(* PLC project variable_speed_drive, Dassault Systèmes ControlBuild 2024x *)
(* stored: creationDateTime 2023-10-03T11:13:08-01:00 *)

(* This module simulates the behaviour of a motor, its variable speed drive and its electrical control logic. The speed setpoint can go from -100% to +100%. *)
FUNCTION_BLOCK equipment_library.variable_speed_drive
  VAR_INPUT
    voltage380 : BOOL := true;
    cmdSupply : BOOL := true;
    sensorSupply : BOOL := true;
  END_VAR
  VAR_INPUT
    forward : BOOL := false;
    speedSetpoint : REAL := 0.0;
  END_VAR
  VAR_OUTPUT
    forwardFB : BOOL := false;
    thermal : BOOL := false;
  END_VAR
  VAR_OUTPUT
    speedVal : REAL := 0.0;
    speedPercent : REAL := 0.0;
  END_VAR
  VAR
    increment : REAL := 0.0;
    memoFwd : BOOL := false;
    forwardState : BOOL := false;
    wantedSpeed : REAL := 0.0;
  END_VAR
  VAR CONSTANT
    nominalSpeed : REAL := 5000.0;
    nominalTime : REAL := 0.5;
    thermalLogic : BOOL := false;
    forwardFbLogic : BOOL := true;
  END_VAR
  VAR
    d_locking : BOOL := false;
    v_d_locking : REAL := 5000.0;
    d_electrical : BOOL := false;
    v_d_electrical : BOOL := false;
    d_forwardFB : BOOL := false;
    v_d_forwardFB : BOOL := false;
  END_VAR


ACTION C_source_code:
/* ----------------------------------------------------------------	*/
/* Type : Model of Operative Behaviour					*/
/* Category :  Associations - motors					*/
/* Author : Dassault Systemes						*/
/* Update date : June 2018							*/
/* ----------------------------------------------------------------	*/
/* This module simulates the behaviour of a motor, its variable	*/
/* speed drive and its electrical control logic.			*/
/* The speed setpoint can go from -100% to +100%.			*/
/* ----------------------------------------------------------------	*/


/* ----------------------------------------------------------------	*/
/* Management of orders from Control Part					*/
/*	if there is no power supply for command 				*/
/*     	the contactors don't understand the control order	*/
/*	The contactors cannot be active in the same time		*/
/*	 	(mechanical security).					*/
/* ----------------------------------------------------------------	*/
if (forward && cmdSupply) memoFwd = 1;
if (!forward || !cmdSupply || d_electrical) memoFwd = 0;


/* ----------------------------------------------------------------	*/
/* Calculation of the on-state of contactor				*/
/* ----------------------------------------------------------------	*/
forwardState= memoFwd & voltage380;

/* ----------------------------------------------------------------	*/
/* Management of the speed ramp						*/
/* ----------------------------------------------------------------	*/
if (d_locking)  speedVal = v_d_locking;
else {
	/* Compute the increment of rotation accoring to the simulation clock */
	if (nominalTime > 0.0)
		increment = (nominalSpeed / nominalTime) * (CLOCK_PERIOD/1000000.0);

	/* Compute the wanted speed according to the speed setpoint	*/
	if (forwardState && (speedSetpoint >= -100.0) &&  (speedSetpoint <= 100.0)) wantedSpeed = (speedSetpoint / 100.0) * nominalSpeed;
	if (! forwardState) wantedSpeed = 0.0;
	
	/* Compute the speed ramp	*/
	if ( speedVal < wantedSpeed ) {
		speedVal += increment;
		if (speedVal > wantedSpeed)  speedVal = wantedSpeed;
	}
	if ( speedVal > wantedSpeed ) {
		speedVal -= increment;
		if (speedVal < wantedSpeed)  speedVal = wantedSpeed;
	}
}

/* ----------------------------------------------------------------	*/
/* Compute the percentage between the current and nominal speed	*/
/* ----------------------------------------------------------------	*/
if (nominalSpeed != 0.0) 
	speedPercent = ((speedVal/nominalSpeed)*100);


/* ----------------------------------------------------------------	*/
/* Management of the thermal feedback					*/
/* ----------------------------------------------------------------	*/
if (d_electrical) thermal=v_d_electrical;
else
	if (sensorSupply) thermal= ! thermalLogic;
	else thermal=0;

/* ----------------------------------------------------------------	*/
/* Management of feedback to Control Part					*/
/*     if a fault is required, the contactor feed-back 		*/
/*		 takes a preset state.					*/
/*	if there is no power supply for sensors 				*/
/*         contactor feed-back returns nothing				*/
/*     else contactor feed-back returns the contactor state combined	*/
/*	    with wiring logic.						*/
/* ----------------------------------------------------------------	*/
if (d_forwardFB) forwardFB=v_d_forwardFB;
else
	if (sensorSupply) forwardFB=(memoFwd ^ ! forwardFbLogic);
	else forwardFB=0;
END_ACTION
END_FUNCTION_BLOCK
